{attribute 'GeneratedUsingTerminal: EPP2817-0008-0016'}
{attribute addProperty BoxType "EPP2817-0008-0016"}
{attribute addProperty Id "Safe_state_activeAT %I*BOOL1Error_channelAT %I*ARRAY[0..2] OF BOOL3Us_UndervoltageAT %I*BOOL1Up_UndervoltageAT %I*BOOL1Sync_errorAT %I*BOOL1TxPDO_ToggleAT %I*BOOL1"}
{attribute addProperty CRC "3987783551"}
{attribute addProperty Size "8"}
TYPE DIG_Inputs_Device_27CCC866 EXTENDS InputBase_8311D824 :
STRUCT
	{attribute addProperty Name "Safe_state_active"}
	Safe_state_active AT %I* : BOOL;
	{attribute addProperty Name "Error_channel"}
	Error_channel AT %I* : ARRAY[0..2] OF BOOL;
	{attribute addProperty Name "Us_Undervoltage"}
	Us_Undervoltage AT %I* : BOOL;
	{attribute addProperty Name "Up_Undervoltage"}
	Up_Undervoltage AT %I* : BOOL;
	{attribute addProperty Name "Sync_error"}
	Sync_error AT %I* : BOOL;
	{attribute addProperty Name "TxPDO_Toggle"}
	TxPDO_Toggle AT %I* : BOOL;
END_STRUCT
END_TYPE

(* stored: Version 1.2.0.0, ProductVersion 3.1.4024.9
   DUT DIG_Inputs_Device_27CCC866: Id {531e6468-37a3-4e28-95a2-5b35d5eb72b5} *)
